// Mitsubishi GX Works2 project: FX1N_Modbus_RTU_V04   PLC: FX1N/FX1NC

PROGRAM MAIN
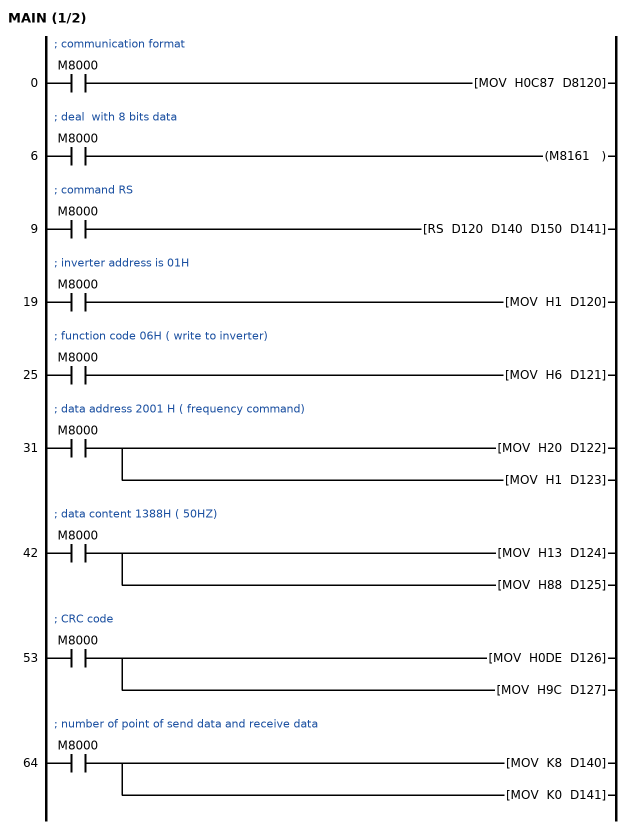
; communication format
0     LD      M8000
      MOV     H0C87 D8120
; deal  with 8 bits data
6     LD      M8000
      OUT     M8161
; command RS
9     LD      M8000
      RS      D120 D140 D150 D141
; inverter address is 01H
19    LD      M8000
      MOV     H1 D120
; function code 06H ( write to inverter)
25    LD      M8000
      MOV     H6 D121
; data address 2001 H ( frequency command)
31    LD      M8000
      MOV     H20 D122
      MOV     H1 D123
; data content 1388H ( 50HZ)
42    LD      M8000
      MOV     H13 D124
      MOV     H88 D125
; CRC code
53    LD      M8000
      MOV     H0DE D126
      MOV     H9C D127
; number of point of send data and receive data
64    LD      M8000
      MOV     K8 D140
      MOV     K0 D141
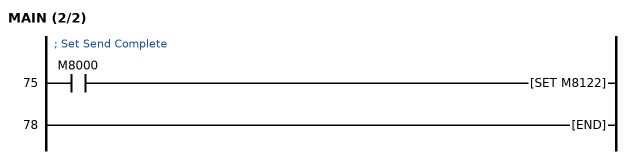
; Set Send Complete
75    LD      M8000
      SET     M8122
78    END
END_PROGRAM
